# EPICS IOC start-up script: iocsh/ethercatmcRawMtrEnc.iocsh
dbLoadRecords("ethercatmcRawMtrEnc.template", "P=$(P), R=$(R), DESC=$(DESC), PREC=$(PREC), MOTOR_PORT=$(MOTOR_PORT), AXIS_NO=$(AXIS_NO)")
